# EPICS StreamDevice protocol: devCombivacApp/Db/test.proto
OutTerminator = CR;
InTerminator = CR;

readPressure{
    out "RPV%(\$1:Channel)d";
    in  "%(\$1:Status)d,\t%g";
}

readVersion{
    out "RVN";
    in  "%f";
}
